// Mitsubishi GX Works2 project: 0625(상하강펄스 회로에넣기)   PLC: Q02/Q02H

PROGRAM MAIN
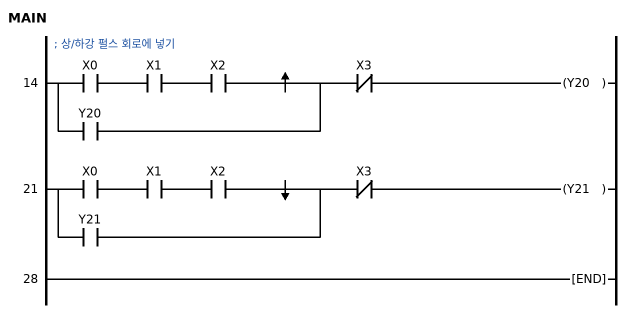
; 상/하강 펄스 회로에 넣기
14    LD      X0
      AND     X1
      AND     X2
      MEP
      OR      Y20
      ANI     X3
      OUT     Y20
21    LD      X0
      AND     X1
      AND     X2
      MEF
      OR      Y21
      ANI     X3
      OUT     Y21
28    END
END_PROGRAM
